// TIA Portal V16 export
// export: Created 2024-10-15T16:30:44.8021566Z, ExportSetting WithDefaults, DisplayName Totally Integrated Automation Portal, DisplayVersion V16, DisplayName TIA Portal Version Control Interface, DisplayVersion V16, DisplayName TIA Portal Openness, DisplayVersion V16, DisplayName STEP 7 Professional, DisplayVersion V16, DisplayName STEP 7 Safety, DisplayVersion V16, DisplayName WinCC Advanced, DisplayVersion V16
DATA_BLOCK "StolyDoCiecia_DB"   // DB4
VERSION : 0.1
// stored: AutoNumber true, InstanceOfName StolyDoCiecia, InstanceOfType FB
"StolyDoCiecia"
BEGIN
END_DATA_BLOCK
